TYPE "Thickness_Measure_Item"
VERSION : 0.1
// Block: Thickness_Measure_Item
   STRUCT
      ID : DInt;
      Time_Stamp : DTL;
      Status : Int;
      Material_Position : LReal;
      Value : Real;
      Err : Real;
      Avg : Real;
      AvgErr : Real;
   END_STRUCT;

END_TYPE
